ADAPTER AStation (* Adapter Interface *)
  (* Standard: 61499-1 *)
  (* Version 1.0, 2018-09-15, az *)
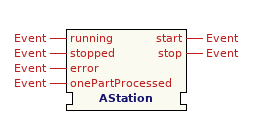
  EVENT_INPUT
    running; (* Request from Socket *)
    stopped;
    error; (* Response from Socket *)
    onePartProcessed;
  END_EVENT
  EVENT_OUTPUT
    start; (* Confirmation from Plug *)
    stop; (* Indication from Plug *)
  END_EVENT
  SERVICE SOCKET/PLUG (* Adapter Interface *)
    SEQUENCE request_confirm
      SOCKET.REQ(REQD) -> PLUG.REQ(REQD);
      PLUG.CNF(CNFD) -> SOCKET.CNF(CNFD);
    END_SEQUENCE
    SEQUENCE indication_response
      PLUG.IND(INDD) -> SOCKET.IND(INDD);
      SOCKET.RSP(RSPD) -> PLUG.RSP(RSPD);
    END_SEQUENCE
  END_SERVICE
END_ADAPTER
